ADAPTER BACnetAdapter (* Adapter Interface *)
  (* Standard: 61499-1 *)
  (* Version 1.0, 2019-10-24, root *)
  (* Compiler header: package fb.test; *)
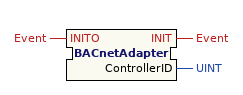
  EVENT_INPUT
    INITO; (* Request from Socket *)
  END_EVENT
  EVENT_OUTPUT
    INIT; (* Confirmation from Plug *)
  END_EVENT
  VAR_OUTPUT
    ControllerID : UINT; (* ID of the Server Controller Instance *)
  END_VAR
END_ADAPTER
